PROGRAM P_CopleyWorkAround
VAR
  bTmp              : BOOL;
  fbTimer           : TON;
  tWait             : TIME := T#6S;
  nIndex, nIdx      : DINT;
  nAxisCount        : DINT := 3;

  aNetId    AT%I*   : AMSNETID;
  nAdr      AT%I*   : ARRAY[1..MAX_AXIS] OF WORD;
  fbEcSetSlaveState : ARRAY[1..MAX_AXIS] OF FB_EcSetSlaveState;

END_VAR
VAR CONSTANT
  MAX_AXIS  : DINT := 10;
END_VAR

nAxisCount := SEL((nAxisCount>MAX_AXIS),nAxisCount,MAX_AXIS);
nAxisCount := SEL((nAxisCount<1),nAxisCount,1);

nIndex := GETCURTASKINDEXEX();
IF _TaskInfo[nIndex].FirstCycle
THEN
  fbTimer.IN := TRUE;
ELSE
  bTmp := TRUE;
  FOR nIdx := 1 TO nAxisCount
  DO
    IF (fbEcSetSlaveState[nIdx].currState.deviceState <> EC_DEVICE_STATE_OP)
    THEN
      bTmp := FALSE;
    END_IF
  END_FOR
  fbTimer.IN := NOT bTmp;
END_IF
fbTimer(PT:= tWait);

FOR nIdx := 1 TO nAxisCount
DO
  fbEcSetSlaveState[nIdx](sNetId:= F_CreateAmsNetId(aNetId), nSlaveAddr:= nAdr[nIdx], bExecute:= fbTimer.Q, reqState:= EC_DEVICE_STATE_OP);
END_FOR

END_PROGRAM

(* stored: Version 1.1.0.1, ProductVersion 3.1.4024.9
   POU P_CopleyWorkAround: Id {e2d7e300-f7b7-4d9b-8f54-701a1ae712fd}, SpecialFunc None *)
